ABB RAPID module: Wobj_wobj_1to1_proto.mod

MODULE Wobj_wobj_1to1_proto
	! Points are read in order of declaration.
  ! Please do not change the order of points!

  LOCAL PERS robtarget pWobj_U_PointX1:=[[2229.307,-198.7225,-777.062],[0.942839741706848,-0.0367999188601971,-0.177168741822243,-0.279839724302292],[-1,1,-2,1],[9E+09,9E+09,9E+09,9E+09,9E+09,9E+09]];
	LOCAL PERS robtarget pWobj_U_PointX2:=[[2398.372,-669.3306,-777.9913],[0.950790882110596,0.10560192912817,-0.152282536029816,-0.248304158449173],[-1,2,-3,1],[9E+09,9E+09,9E+09,9E+09,9E+09,9E+09]];
	LOCAL PERS robtarget pWobj_U_PointY1:=[[1636.653,-736.9378,-776.6005],[0.95078980922699,0.105600602924824,-0.152329280972481,-0.248280212283134],[-1,2,-4,1],[9E+09,9E+09,9E+09,9E+09,9E+09,9E+09]];

ENDMODULE
